FUNCTION_BLOCK SS3_PnP (* Basic FB with empty ECC *)
  (* Standard: 61499-2 *)
  (* Version 1.0, 2025-08-24, DEVIASH *)
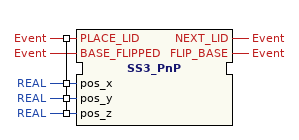
  EVENT_INPUT
    PLACE_LID WITH pos_x, pos_y, pos_z;
    BASE_FLIPPED;
  END_EVENT
  EVENT_OUTPUT
    NEXT_LID;
    FLIP_BASE;
  END_EVENT
  VAR_INPUT
    pos_x : REAL;
    pos_y : REAL;
    pos_z : REAL;
  END_VAR
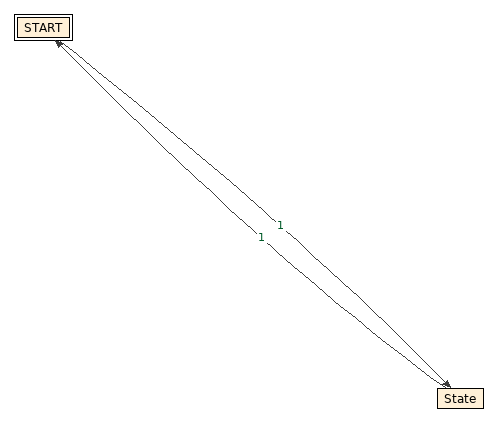
  EC_STATES
    START; (* Initial State *)
    State;
  END_STATES
  EC_TRANSITIONS
    START TO State := 1;
    State TO START := 1;
  END_TRANSITIONS
END_FUNCTION_BLOCK
